FUNCTION_BLOCK Wago1405_6 (* Service Interface Function Block Type *)
  (* Standard: 61499-2; Description: Copyright (c) 2018, 2024 fortiss GmbH This program and the accompanying materials are made available under the terms of the Eclipse Public License 2.0 which is available at https://www.eclipse.org/legal/epl-2.0/ SPDX-License-Identifier: EPL-2.0 *)
  (* Version 1.0, 2018-12-05, Jose Cabral *)
  (* Version 1.1, 2024-09-22, Monika Wenger *)
  (* Version 3.0, 2025-04-14, Patrick Aigner, changed package *)
  PACKAGE eclipse4diac::io::wago;
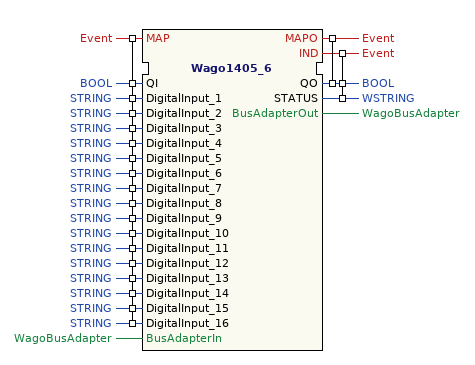
  EVENT_INPUT
    MAP WITH DigitalInput_1, DigitalInput_2, DigitalInput_5, DigitalInput_3, DigitalInput_4, DigitalInput_6, DigitalInput_7, DigitalInput_8, DigitalInput_9, DigitalInput_10, DigitalInput_11, DigitalInput_12, DigitalInput_13, DigitalInput_14, DigitalInput_15, DigitalInput_16, QI; (* Map Pins *)
  END_EVENT
  EVENT_OUTPUT
    MAPO WITH QO; (* Confirm Pin Mapping *)
    IND WITH QO, STATUS; (* Indication from Resource *)
  END_EVENT
  VAR_INPUT
    QI : BOOL; (* Event Input Qualifier *)
    DigitalInput_1 : STRING;
    DigitalInput_2 : STRING;
    DigitalInput_3 : STRING;
    DigitalInput_4 : STRING;
    DigitalInput_5 : STRING;
    DigitalInput_6 : STRING;
    DigitalInput_7 : STRING;
    DigitalInput_8 : STRING;
    DigitalInput_9 : STRING;
    DigitalInput_10 : STRING;
    DigitalInput_11 : STRING;
    DigitalInput_12 : STRING;
    DigitalInput_13 : STRING;
    DigitalInput_14 : STRING;
    DigitalInput_15 : STRING;
    DigitalInput_16 : STRING;
  END_VAR
  VAR_OUTPUT
    QO : BOOL; (* Event Output Qualifier *)
    STATUS : WSTRING; (* Service Status *)
  END_VAR
  SOCKETS
    BusAdapterIn : eclipse4diac::io::wago::WagoBusAdapter;
  END_SOCKETS
  PLUGS
    BusAdapterOut : eclipse4diac::io::wago::WagoBusAdapter;
  END_PLUGS
END_FUNCTION_BLOCK
